(* IEC 61131-3 sources: POMIRTS_lab3/AS/Library/AsXml, 3 files *)

(* ---- AsXml.typ ---- *)
(********************************************************************
 * COPYRIGHT -- Bernecker + Rainer
 ********************************************************************
 * Library: AsXml
 * File: AsXml.typ
 * Author: B+R
 ********************************************************************
 * Data types of library AsXml
 ********************************************************************)

TYPE

END_TYPE

(* ---- AsXml.fun ---- *)
(********************************************************************
 * COPYRIGHT -- Bernecker + Rainer
 ********************************************************************
 * Library: AsXml
 * File: AsXml.fun
 * Author: B+R
 ********************************************************************
 * Functions and function blocks of library AsXml
 ********************************************************************)

FUNCTION_BLOCK xmlCreateMemoryReader	(*creates an xml memory reader*)
	VAR_INPUT
		enable			: BOOL;			(*enables execution*)
		pXmlMemory		: UDINT;		(*pointer to the XML data*)
		memorySize		: UDINT;		(*size of the XML data*)
	END_VAR

	VAR_OUTPUT
		status			: UINT;			(*execution status: ERR_OK, ERR_FUB_ENABLE_FALSE, ERR_FUB_BUSY, 0xXXXX = see help*)
		ident			: UDINT;		(*identifier*)
	END_VAR
END_FUNCTION_BLOCK

FUNCTION_BLOCK xmlCloseMemoryReader		(*closes the xml memory reader*)
	VAR_INPUT
		enable			: BOOL;			(*enables execution*)
		ident			: UDINT;		(*identifier*)
	END_VAR

	VAR_OUTPUT
		status			: UINT;			(*execution status: ERR_OK, ERR_FUB_ENABLE_FALSE, ERR_FUB_BUSY, 0xXXXX = see help*)
	END_VAR
END_FUNCTION_BLOCK

FUNCTION_BLOCK xmlReadNextNode			(*reads the next XML node*)
	VAR_INPUT
		enable			: BOOL;			(*enables execution*)
		ident			: UDINT;		(*identifier*)
		forceRead		: BOOL;			(*reads next Node even if last node could not be read successfully*)
		skipSubtree		: BOOL;			(*avoids XML nodes in the subtree*)
		pName			: UDINT;		(*pointer to buffer for the XML node name*)
		nameSize		: UDINT;		(*size of the buffer for the XML node name*)
		pValue			: UDINT;		(*pointer to buffer for the XML node value*)
		valueSize		: UDINT;		(*size of the buffer for the XML node value*)
	END_VAR

	VAR_OUTPUT
		status			: UINT;			(*execution status: ERR_OK, ERR_FUB_ENABLE_FALSE, ERR_FUB_BUSY, 0xXXXX = see help*)
		nodeType		: UDINT;		(*type of the XML node*)
		depth			: UDINT;		(*depth of the XML node*)
		isEmpty			: BOOL;			(*empty XML node?*)
		attributeCount	: UDINT;		(*number of attributes*)
		neededNameSize	: UDINT;		(*needed name buffer size*)
		neededValueSize	: UDINT;		(*needed value buffer size*)
	END_VAR
END_FUNCTION_BLOCK

FUNCTION_BLOCK xmlReadAttributeNr		(*reads the next attribute of the XML node*)
	VAR_INPUT
		enable			: BOOL;			(*enables execution*)
		ident			: UDINT;		(*identifier*)
		index			: UDINT;		(*index of the attribute to read*)
		pName			: UDINT;		(*pointer to buffer for the attribute name*)
		nameSize		: UDINT;		(*size of the buffer for the XML attribute name*)
		pValue			: UDINT;		(*pointer to buffer for the attribute value*)
		valueSize		: UDINT;		(*size of the buffer for the XML attribute value*)
	END_VAR

	VAR_OUTPUT
		status			: UINT;			(*execution status: ERR_OK, ERR_FUB_ENABLE_FALSE, ERR_FUB_BUSY, 0xXXXX = see help*)
		neededNameSize	: UDINT;		(*needed name buffer size*)
		neededValueSize	: UDINT;		(*needed value buffer size*)
	END_VAR
END_FUNCTION_BLOCK

FUNCTION_BLOCK xmlCreateMemoryWriter	(*creates an xml memory writer*)
	VAR_INPUT
		enable			: BOOL;			(*enables execution*)
	END_VAR

	VAR_OUTPUT
		status			: UINT;			(*execution status: ERR_OK, ERR_FUB_ENABLE_FALSE, ERR_FUB_BUSY, 0xXXXX = see help*)
		ident			: UDINT;		(*identifier*)
	END_VAR
END_FUNCTION_BLOCK

FUNCTION_BLOCK xmlGetMemoryInfo			(*gets the pointer to and the size of the created XML data*)
	VAR_INPUT
		enable			: BOOL;			(*enables execution*)
		ident			: UDINT;		(*identifier*)
	END_VAR

	VAR_OUTPUT
		status			: UINT;			(*execution status: ERR_OK, ERR_FUB_ENABLE_FALSE, 0xXXXX = see help*)
		pXmlData		: UDINT;		(*pointer to the created XML data*)
		xmlDataSize		: UDINT;		(*size of the created XML data*)
	END_VAR
END_FUNCTION_BLOCK

FUNCTION_BLOCK xmlCloseMemoryWriter		(*closes the xml memory writer and releases the allocated memory*)
	VAR_INPUT
		enable			: BOOL;			(*enables execution*)
		ident			: UDINT;		(*identifier*)
	END_VAR

	VAR_OUTPUT
		status			: UINT;			(*execution status: ERR_OK, ERR_FUB_ENABLE_FALSE, ERR_FUB_BUSY, 0xXXXX = see help*)
	END_VAR
END_FUNCTION_BLOCK

FUNCTION_BLOCK xmlWriteStartDocument	(*writes the version and the encoding of the document*)
	VAR_INPUT
		enable			: BOOL;			(*enables execution*)
		ident			: UDINT;		(*identifier*)
		pVersion		: UDINT;		(*pointer to the version*)
		pEncoding		: UDINT;		(*pointer to the encoding*)
		pStandalone		: UDINT;		(*pointer to the standalone text*)
	END_VAR

	VAR_OUTPUT
		status			: UINT;			(*execution status: ERR_OK, ERR_FUB_ENABLE_FALSE, ERR_FUB_BUSY, 0xXXXX = see help*)
	END_VAR
END_FUNCTION_BLOCK

FUNCTION_BLOCK xmlWriteEndDocument		(*finishes the document*)
	VAR_INPUT
		enable			: BOOL;			(*enables execution*)
		ident			: UDINT;		(*identifier*)
	END_VAR

	VAR_OUTPUT
		status			: UINT;			(*execution status: ERR_OK, ERR_FUB_ENABLE_FALSE, ERR_FUB_BUSY, 0xXXXX = see help*)
	END_VAR
END_FUNCTION_BLOCK

FUNCTION_BLOCK xmlWriteStartElement		(*starts a new XML element*)
	VAR_INPUT
		enable			: BOOL;			(*enables execution*)
		ident			: UDINT;		(*identifier*)
		pName			: UDINT;		(*pointer to the XML element name*)
	END_VAR

	VAR_OUTPUT
		status			: UINT;			(*execution status: ERR_OK, ERR_FUB_ENABLE_FALSE, ERR_FUB_BUSY, 0xXXXX = see help*)
	END_VAR
END_FUNCTION_BLOCK

FUNCTION_BLOCK xmlWriteAttribute		(*adds an attribute to the current XML element*)
	VAR_INPUT
		enable			: BOOL;			(*enables execution*)
		ident			: UDINT;		(*identifier*)
		pName			: UDINT;		(*pointer to the XML attribute name*)
		pValue			: UDINT;		(*pointer to the XML attribute value*)
	END_VAR

	VAR_OUTPUT
		status			: UINT;			(*execution status: ERR_OK, ERR_FUB_ENABLE_FALSE, ERR_FUB_BUSY, 0xXXXX = see help*)
	END_VAR
END_FUNCTION_BLOCK

FUNCTION_BLOCK xmlWriteElementText		(*writes an XML element text*)
	VAR_INPUT
		enable			: BOOL;			(*enables execution*)
		ident			: UDINT;		(*identifier*)
		pText			: UDINT;		(*pointer to the element text*)
	END_VAR

	VAR_OUTPUT
		status			: UINT;			(*execution status: ERR_OK, ERR_FUB_ENABLE_FALSE, ERR_FUB_BUSY, 0xXXXX = see help*)
	END_VAR
END_FUNCTION_BLOCK

FUNCTION_BLOCK xmlWriteEndElement		(*closes the current XML element*)
	VAR_INPUT
		enable			: BOOL;			(*enables execution*)
		ident			: UDINT;		(*identifier*)
	END_VAR

	VAR_OUTPUT
		status			: UINT;			(*execution status: ERR_OK, ERR_FUB_ENABLE_FALSE, ERR_FUB_BUSY, 0xXXXX = see help*)
	END_VAR
END_FUNCTION_BLOCK

FUNCTION_BLOCK xmlWriteComment			(*writes an XML comment*)
	VAR_INPUT
		enable			: BOOL;			(*enables execution*)
		ident			: UDINT;		(*identifier*)
		pText			: UDINT;		(*pointer to the comment text*)
	END_VAR

	VAR_OUTPUT
		status			: UINT;			(*execution status: ERR_OK, ERR_FUB_ENABLE_FALSE, ERR_FUB_BUSY, 0xXXXX = see help*)
	END_VAR
END_FUNCTION_BLOCK

FUNCTION_BLOCK xmlWriteCData			(*writes an XML CDATA Section*)
	VAR_INPUT
		enable			: BOOL;			(*enables execution*)
		ident			: UDINT;		(*identifier*)
		pCData			: UDINT;		(*pointer to the CDATA data*)
	END_VAR

	VAR_OUTPUT
		status			: UINT;			(*execution status: ERR_OK, ERR_FUB_ENABLE_FALSE, ERR_FUB_BUSY, 0xXXXX = see help*)
	END_VAR
END_FUNCTION_BLOCK

FUNCTION_BLOCK xmlWritePI				(*writes an XML process instruction*)
	VAR_INPUT
		enable			: BOOL;			(*enables execution*)
		ident			: UDINT;		(*identifier*)
		pTarget			: UDINT;		(*pointer to the process instruction*)
		pValue			: UDINT;		(*pointer to the pi value*)
	END_VAR

	VAR_OUTPUT
		status			: UINT;			(*execution status: ERR_OK, ERR_FUB_ENABLE_FALSE, ERR_FUB_BUSY, 0xXXXX = see help*)
	END_VAR
END_FUNCTION_BLOCK

(* ---- AsXml.var ---- *)
(********************************************************************
 * COPYRIGHT -- Bernecker + Rainer
 ********************************************************************
 * Library: AsXml
 * File: AsXml.var
 * Author: B+R
 ********************************************************************
 * Local variables of library AsXml
 ********************************************************************)

VAR CONSTANT
	xmlERR_MEMORY		    	: UINT		:= 33810;	(*memory error*)
	xmlERR_INVALID_PARAMETER	: UINT		:= 33811;	(*wrong parameter or nullpointer given*)
	xmlERR_GENERAL				: UINT		:= 33812;  	(*general XML error*)
	xmlERR_NO_FURTHER_XML_NODE	: UINT		:= 33813; 	(*no further XML node available*)
	xmlERR_NAME_BUFFER_TOO_SMALL: UINT		:= 33814; 	(*buffer for name too small*)
	xmlERR_VALUE_BUFFER_TOO_SMALL: UINT		:= 33815; 	(*buffer for value too small*)
	xmlERR_INVALID_ATTRIBUTE_INDEX: UINT	:= 33816; 	(*invalid attribute index*)
	xmlERR_NO_ATTRIBUTES		: UINT		:= 33817; 	(*no attribute available*)
	xmlERR_XML_DATA_INVALID		: UINT		:= 33818; 	(*xml data is invalid*)
	xmlERR_INVALID_IDENT 		: UINT		:= 33819;	(*error identifier invalid*)
	xmlERR_NO_ELEMENT_OPEN		: UINT		:= 33820; 	(*no open XML element where to put the attribute*)
	xmlERR_INVALID_POSITION		: UINT		:= 33821;	(*invalid position for this node*)
	xmlERR_CONVERT				: UINT		:= 33822;	(*error during converting text*)
	xmlERR_CONVERT_TEXT			: UINT   	:= 33823;	(*error converting text*)
	xmlERR_UNSUPPORTED_ENCODING : UINT		:= 33824;	(*unsupported encoding*)

	xmlNODE_TYPE_ELEMENT		: UINT		:= 1;		(*XML element node*)
	xmlNODE_TYPE_TEXT			: UINT		:= 3;		(*XML element text*)
	xmlNODE_TYPE_CDATA			: UINT		:= 4;		(*XML CDATA section*)
	xmlNODE_TYPE_PI				: UINT		:= 7;		(*XML process instruction node*)
	xmlNODE_TYPE_COMMENT		: UINT		:= 8;		(*XML comment*)
	xmlNODE_TYPE_WHITESPACE		: UINT		:= 13;		(*XML white space*)
	xmlNODE_TYPE_SIGN_WHITESPACE: UINT		:= 14;		(*XML significant white space*)
	xmlNODE_TYPE_ENDELEMENT		: UINT		:= 15;		(*XML end element node*)
END_VAR
